PROGRAM Axis02_Speed_Offset
VAR
END_VAR

END_PROGRAM

(* stored: Version 1.1.0.1, ProductVersion 3.1.4024.15
   POU Axis02_Speed_Offset: Id {2cbf813d-8b48-47d1-9152-8ba7814b17f0}, SpecialFunc None *)
